// TwinCAT 3 PLC project PLC1
// ProgramVersion: 3.1.4024.0
// libraries:
//   Tc2_Standard, * (Beckhoff Automation GmbH)
//   Tc2_System, * (Beckhoff Automation GmbH)
//   Tc3_Module, * (Beckhoff Automation GmbH)
// project tree:
//   / PlcTask.TcTTO
//   POUs/ MAIN.TcPOU
// real-time tasks:
//   TASK PlcTask: cycle T#5ms, priority 20, ADS port 350
// I/O:
//   DEVICE Device 1 (EtherCAT Simulation), AmsNetId 10.33.70.115.2.1
//     Term 1 (EK1100) // EK1100-0000-0018
//     Term 2 (EL1512) // EL1512-0000-0021
//     Term 3 (EL2008) // EL2008-0000-0018
// variable links:
//   PLC1/PLC1 Instance <-> Device 1 (EtherCAT Simulation)
//     PlcTask Inputs/MAIN.ecat_sim_device_state <-> Inputs/DevState

CONFIGURATION PLC1
    RESOURCE PLC ON TwinCAT3
        TASK PlcTask(INTERVAL := T#5ms, PRIORITY := 20);
        PROGRAM MAIN WITH PlcTask : MAIN;
    END_RESOURCE
END_CONFIGURATION

// ---- POUs/MAIN.TcPOU
PROGRAM MAIN
VAR
	ecat_sim_device_state AT %I* : UINT;
END_VAR

END_PROGRAM
